PROGRAM Stn8
VAR

	start8: BOOL;
	reset8: BOOL;

	Stn8ProcessFE: F_TRIG;
	Stn8ProcessRE: R_TRIG;
	bCutStn8ProcessHalt: BOOL;
	DoorClose8: R_TRIG;
	bStn8DoorClamp: BOOL;

END_VAR

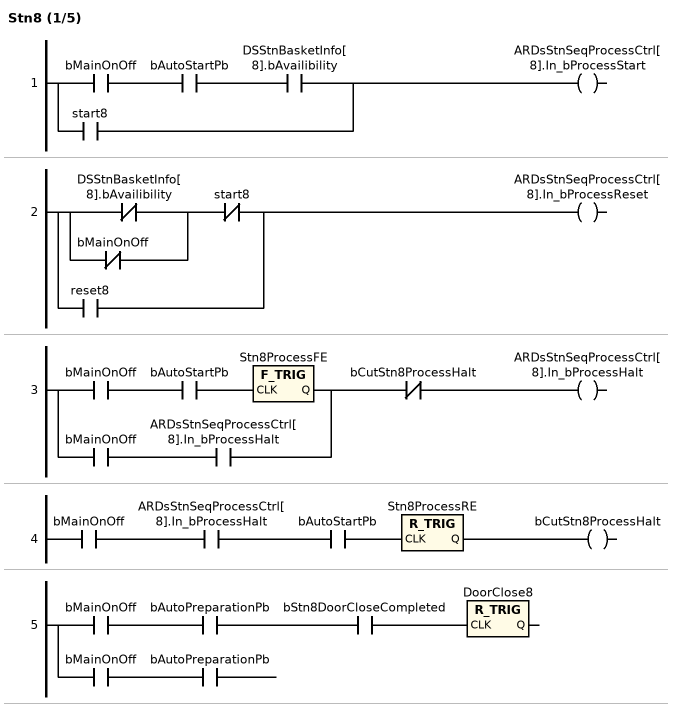
// NETWORK 1
ARDsStnSeqProcessCtrl[8].In_bProcessStart := bMainOnOff AND bAutoStartPb AND DSStnBasketInfo[8].bAvailibility OR start8;

// NETWORK 2
ARDsStnSeqProcessCtrl[8].In_bProcessReset := (NOT DSStnBasketInfo[8].bAvailibility OR NOT bMainOnOff) AND NOT start8 OR reset8;

// NETWORK 3
Stn8ProcessFE(CLK := bMainOnOff AND bAutoStartPb); // F_TRIG
ARDsStnSeqProcessCtrl[8].In_bProcessHalt := (Stn8ProcessFE.Q OR bMainOnOff AND ARDsStnSeqProcessCtrl[8].In_bProcessHalt) AND NOT bCutStn8ProcessHalt;

// NETWORK 4
Stn8ProcessRE(CLK := bMainOnOff AND ARDsStnSeqProcessCtrl[8].In_bProcessHalt AND bAutoStartPb); // R_TRIG
bCutStn8ProcessHalt := Stn8ProcessRE.Q;

// NETWORK 5
DoorClose8(CLK := bMainOnOff AND bAutoPreparationPb AND bStn8DoorCloseCompleted); // R_TRIG
(* DoorClose8.Q OR bMainOnOff AND bAutoPreparationPb; result not used *)

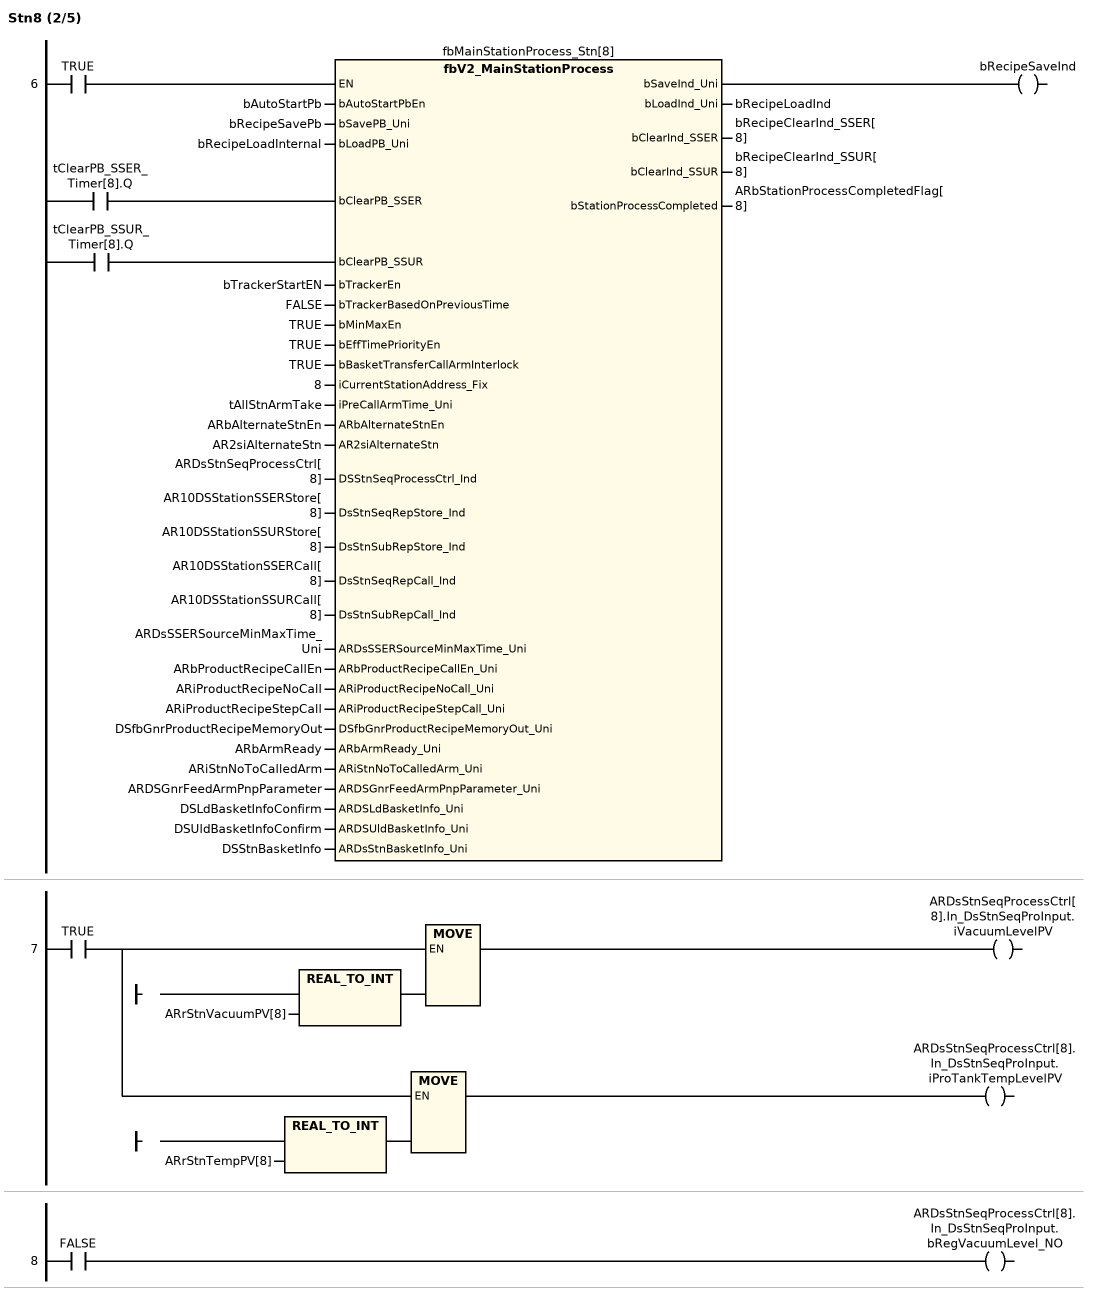
// NETWORK 6
fbMainStationProcess_Stn[8](
    bAutoStartPbEn := bAutoStartPb,
    bSavePB_Uni := bRecipeSavePb,
    bLoadPB_Uni := bRecipeLoadInternal,
    bClearPB_SSER := tClearPB_SSER_Timer[8].Q,
    bClearPB_SSUR := tClearPB_SSUR_Timer[8].Q,
    bTrackerEn := bTrackerStartEN,
    bTrackerBasedOnPreviousTime := FALSE,
    bMinMaxEn := TRUE,
    bEffTimePriorityEn := TRUE,
    bBasketTransferCallArmInterlock := TRUE,
    iCurrentStationAddress_Fix := 8,
    iPreCallArmTime_Uni := tAllStnArmTake,
    ARbAlternateStnEn := ARbAlternateStnEn,
    AR2siAlternateStn := AR2siAlternateStn,
    DSStnSeqProcessCtrl_Ind := ARDsStnSeqProcessCtrl[8],
    DsStnSeqRepStore_Ind := AR10DSStationSSERStore[8],
    DsStnSubRepStore_Ind := AR10DSStationSSURStore[8],
    DsStnSeqRepCall_Ind := AR10DSStationSSERCall[8],
    DsStnSubRepCall_Ind := AR10DSStationSSURCall[8],
    ARDsSSERSourceMinMaxTime_Uni := ARDsSSERSourceMinMaxTime_Uni,
    ARbProductRecipeCallEn_Uni := ARbProductRecipeCallEn,
    ARiProductRecipeNoCall_Uni := ARiProductRecipeNoCall,
    ARiProductRecipeStepCall_Uni := ARiProductRecipeStepCall,
    DSfbGnrProductRecipeMemoryOut_Uni := DSfbGnrProductRecipeMemoryOut,
    ARbArmReady_Uni := ARbArmReady,
    ARiStnNoToCalledArm_Uni := ARiStnNoToCalledArm,
    ARDSGnrFeedArmPnpParameter_Uni := ARDSGnrFeedArmPnpParameter,
    ARDSLdBasketInfo_Uni := DSLdBasketInfoConfirm,
    ARDSUldBasketInfo_Uni := DSUldBasketInfoConfirm,
    ARDsStnBasketInfo_Uni := DSStnBasketInfo,
    bLoadInd_Uni => bRecipeLoadInd,
    bClearInd_SSER => bRecipeClearInd_SSER[8],
    bClearInd_SSUR => bRecipeClearInd_SSUR[8],
    bStationProcessCompleted => ARbStationProcessCompletedFlag[8]); // fbV2_MainStationProcess
bRecipeSaveInd := fbMainStationProcess_Stn[8].bSaveInd_Uni;

// NETWORK 7
ARDsStnSeqProcessCtrl[8].In_DsStnSeqProInput.iVacuumLevelPV := REAL_TO_INT(ARrStnVacuumPV[8]);
ARDsStnSeqProcessCtrl[8].In_DsStnSeqProInput.iProTankTempLevelPV := REAL_TO_INT(ARrStnTempPV[8]);

// NETWORK 8
ARDsStnSeqProcessCtrl[8].In_DsStnSeqProInput.bRegVacuumLevel_NO := FALSE;

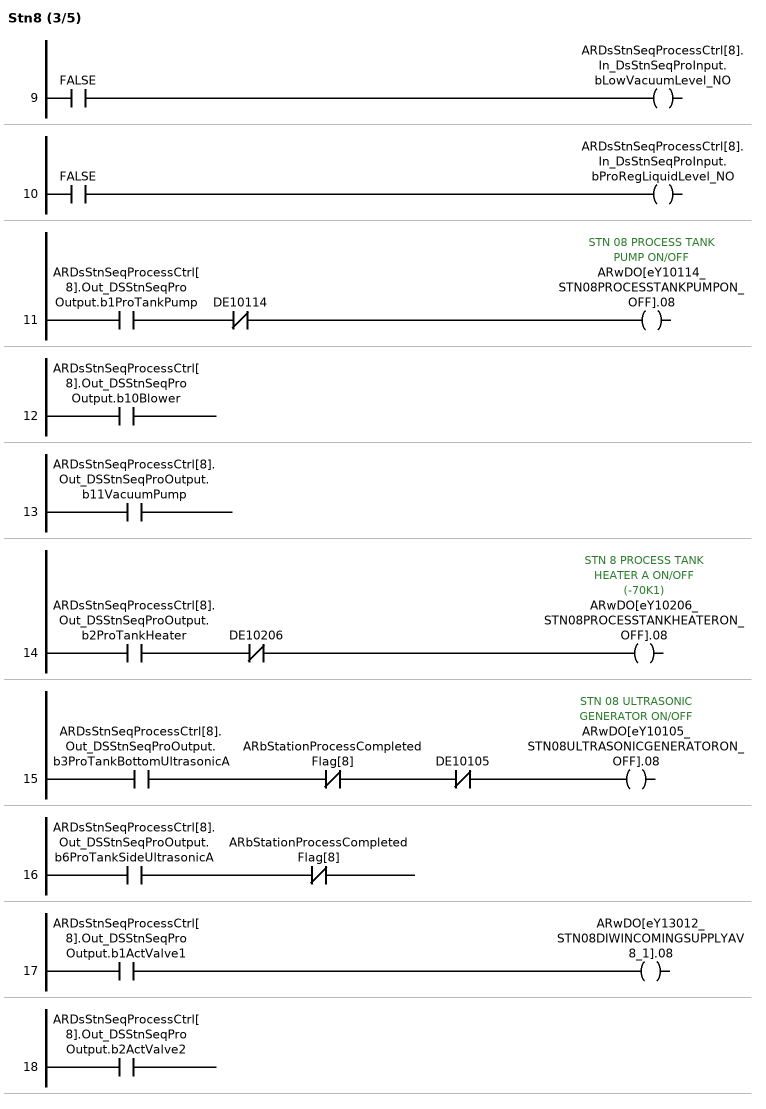
// NETWORK 9
ARDsStnSeqProcessCtrl[8].In_DsStnSeqProInput.bLowVacuumLevel_NO := FALSE;

// NETWORK 10
ARDsStnSeqProcessCtrl[8].In_DsStnSeqProInput.bProRegLiquidLevel_NO := FALSE;

// NETWORK 11
//   ARwDO[eY10114_STN08PROCESSTANKPUMPON_OFF].08: STN 08 PROCESS TANK PUMP ON/OFF
ARwDO[eY10114_STN08PROCESSTANKPUMPON_OFF].08 := ARDsStnSeqProcessCtrl[8].Out_DSStnSeqProOutput.b1ProTankPump AND NOT DE10114;

// NETWORK 12
(* ARDsStnSeqProcessCtrl[8].Out_DSStnSeqProOutput.b10Blower; not connected *)

// NETWORK 13
(* ARDsStnSeqProcessCtrl[8].Out_DSStnSeqProOutput.b11VacuumPump; not connected *)

// NETWORK 14
//   ARwDO[eY10206_STN08PROCESSTANKHEATERON_OFF].08: STN 8 PROCESS TANK HEATER A ON/OFF (-70K1)
ARwDO[eY10206_STN08PROCESSTANKHEATERON_OFF].08 := ARDsStnSeqProcessCtrl[8].Out_DSStnSeqProOutput.b2ProTankHeater AND NOT DE10206;

// NETWORK 15
//   ARwDO[eY10105_STN08ULTRASONICGENERATORON_OFF].08: STN 08 ULTRASONIC GENERATOR ON/OFF
ARwDO[eY10105_STN08ULTRASONICGENERATORON_OFF].08 := ARDsStnSeqProcessCtrl[8].Out_DSStnSeqProOutput.b3ProTankBottomUltrasonicA AND NOT ARbStationProcessCompletedFlag[8] AND NOT DE10105;

// NETWORK 16
(* ARDsStnSeqProcessCtrl[8].Out_DSStnSeqProOutput.b6ProTankSideUltrasonicA AND NOT ARbStationProcessCompletedFlag[8]; result not used *)

// NETWORK 17
ARwDO[eY13012_STN08DIWINCOMINGSUPPLYAV8_1].08 := ARDsStnSeqProcessCtrl[8].Out_DSStnSeqProOutput.b1ActValve1;

// NETWORK 18
(* ARDsStnSeqProcessCtrl[8].Out_DSStnSeqProOutput.b2ActValve2; not connected *)

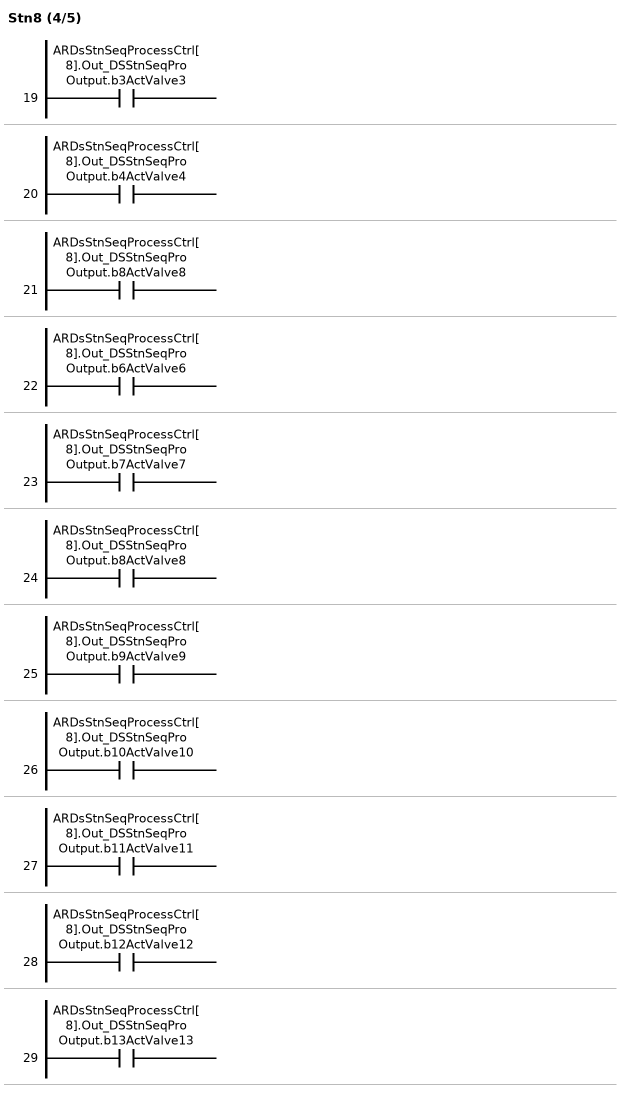
// NETWORK 19
(* ARDsStnSeqProcessCtrl[8].Out_DSStnSeqProOutput.b3ActValve3; not connected *)

// NETWORK 20
(* ARDsStnSeqProcessCtrl[8].Out_DSStnSeqProOutput.b4ActValve4; not connected *)

// NETWORK 21
(* ARDsStnSeqProcessCtrl[8].Out_DSStnSeqProOutput.b8ActValve8; not connected *)

// NETWORK 22
(* ARDsStnSeqProcessCtrl[8].Out_DSStnSeqProOutput.b6ActValve6; not connected *)

// NETWORK 23
(* ARDsStnSeqProcessCtrl[8].Out_DSStnSeqProOutput.b7ActValve7; not connected *)

// NETWORK 24
(* ARDsStnSeqProcessCtrl[8].Out_DSStnSeqProOutput.b8ActValve8; not connected *)

// NETWORK 25
(* ARDsStnSeqProcessCtrl[8].Out_DSStnSeqProOutput.b9ActValve9; not connected *)

// NETWORK 26
(* ARDsStnSeqProcessCtrl[8].Out_DSStnSeqProOutput.b10ActValve10; not connected *)

// NETWORK 27
(* ARDsStnSeqProcessCtrl[8].Out_DSStnSeqProOutput.b11ActValve11; not connected *)

// NETWORK 28
(* ARDsStnSeqProcessCtrl[8].Out_DSStnSeqProOutput.b12ActValve12; not connected *)

// NETWORK 29
(* ARDsStnSeqProcessCtrl[8].Out_DSStnSeqProOutput.b13ActValve13; not connected *)

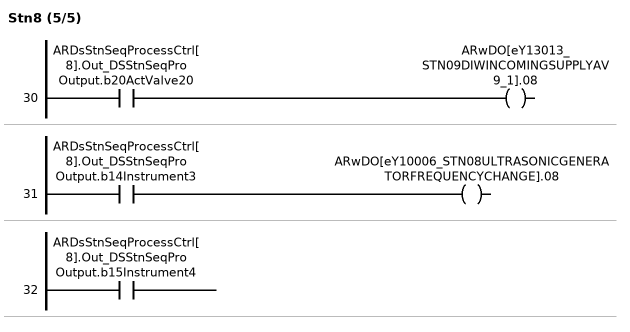
// NETWORK 30
ARwDO[eY13013_STN09DIWINCOMINGSUPPLYAV9_1].08 := ARDsStnSeqProcessCtrl[8].Out_DSStnSeqProOutput.b20ActValve20;

// NETWORK 31
ARwDO[eY10006_STN08ULTRASONICGENERATORFREQUENCYCHANGE].08 := ARDsStnSeqProcessCtrl[8].Out_DSStnSeqProOutput.b14Instrument3;

// NETWORK 32
(* ARDsStnSeqProcessCtrl[8].Out_DSStnSeqProOutput.b15Instrument4; not connected *)

END_PROGRAM

(* stored: Version 1.1.0.1, ProductVersion 3.1.4024.12
   POU Stn8: Id {1c4dd3f5-32c3-4b15-9952-195b8291cab4}, SpecialFunc None *)
